PROGRAM PRG_RunTests
VAR
    fbRangeComparison : FB_TestRangeComparison;
    fbShutterSafety : FB_TestShutterSafety;
	fbCentroidTest : FB_Test_EpicsCentroidMonitor;
    fbMotorTest : FB_Test_EpicsMotorMonitor;

END_VAR

TcUnit.RUN();

END_PROGRAM

(* stored: Version 1.1.0.1, ProductVersion 3.1.4022.18
   POU PRG_RunTests: Id {ad02aa03-9ff9-4ff4-bd78-c8e4c4fadc0f}, SpecialFunc None *)
